{attribute 'linkalways'} 
{attribute 'no_explicit_call' := 'This FB is a CLASS and must be accessed using methods or properties'}
{attribute 'enable_dynamic_creation'}
FUNCTION_BLOCK LinkedListChangedEvent EXTENDS Disposable IMPLEMENTS I_LinkedListChangedEvent
VAR
	_targetLinkedList : I_LinkedList;
END_VAR

METHOD FB_init : BOOL
VAR_INPUT
	bInitRetains : BOOL; // if TRUE, the retain variables are initialized (warm start / cold start)
	bInCopyCode : BOOL;  // if TRUE, the instance afterwards gets moved into the copy code (online change)
	TargetLinkedList : I_LinkedList;
END_VAR
This^._targetLinkedList := TargetLinkedList;
END_METHOD

PROPERTY PUBLIC TargetLinkedList : I_LinkedList
GET // PUBLIC
TargetLinkedList := _targetLinkedList;
END_GET
END_PROPERTY

END_FUNCTION_BLOCK

(* stored: Version 1.1.0.1, ProductVersion 3.1.4024.12
   POU LinkedListChangedEvent: Id {9610cf6e-6a94-4041-a95d-cecc28a7cd91}, SpecialFunc None
   Folder Constructor: Id {96f7420d-ef8b-4a36-bac7-923e9ebf4e3c}
   Method FB_init: Id {a156c7fb-49bc-41cc-8bf0-976196f15949}
   Property TargetLinkedList: Id {af9c3577-5c7c-47cf-b981-2d76dda3372a}
   Get Get: Id {02433bd2-0877-4583-83d2-4366515e4d88} *)
